FUNCTION_BLOCK Clock IMPLEMENTS Cyclic
VAR
	_Enable : BOOL;
	_Period : TIME;
	_Duty : LREAL := 0.5;
	switchTime : TIME;
	timer : TON;
	_Clock : BOOL;
END_VAR

METHOD PRIVATE CalcSwitchTime
switchTime := LREAL_TO_TIME(TIME_TO_LREAL(_Period) * _Duty);
END_METHOD

{attribute 'monitoring' := 'call'}
PROPERTY Clock : BOOL
GET
Clock := _Clock;
END_GET
END_PROPERTY

METHOD Cyclic
timer(IN := _Enable, PT := _Period);
IF (timer.Q) THEN
	timer(IN := FALSE);
	timer(IN := TRUE);
END_IF
_Clock := _Enable AND timer.ET >= switchTime;
END_METHOD

{attribute 'monitoring' := 'call'}
PROPERTY Duty : LREAL
GET
Duty := _Duty;
END_GET
SET
_Duty := Duty;
CalcSwitchTime();
END_SET
END_PROPERTY

{attribute 'monitoring' := 'call'}
PROPERTY Enable : BOOL
GET
Enable := _Enable;
END_GET
SET
_Enable := Enable;
END_SET
END_PROPERTY

{attribute 'monitoring' := 'call'}
PROPERTY Frequency : LREAL
GET
IF (_Period > T#0S) THEN
	Frequency := 1000/TIME_TO_LREAL(_Period);
ELSE
	Frequency := 0;
END_IF
END_GET
SET
IF (Frequency > 0) THEN
	_Period := LREAL_TO_TIME(1000/Frequency);
ELSE
	_Period := T#0S;
END_IF
CalcSwitchTime();
END_SET
END_PROPERTY

{attribute 'monitoring' := 'call'}
PROPERTY Period : TIME
GET
Period := _Period;
END_GET
SET
_Period := Period;
CalcSwitchTime();
END_SET
END_PROPERTY

END_FUNCTION_BLOCK

(* stored: Version 1.1.0.1
   POU Clock: Id {12e9d754-7a2e-04e4-151b-81bf53a123a4}, SpecialFunc None
   Method CalcSwitchTime: Id {eeb3fa65-90da-0834-10c0-64a9d6b20f5f}
   Property Clock: Id {94afcf8c-3fec-03bf-0ea5-551f99fbc25b}
   Get Get: Id {86ccfb57-1f88-0117-3a6c-95826046587c}
   Method Cyclic: Id {d126b246-8ccf-0404-1dbe-459eed47bff6}
   Property Duty: Id {62ad35f6-8917-03d8-1e82-2f52ccf6ca78}
   Get Get: Id {8de1ac67-05b7-0036-0652-56a889ec5cee}
   Set Set: Id {3b362bf6-5c6f-0809-0f27-e988aae87027}
   Property Enable: Id {6422a66f-fc11-03a1-3de3-f3d118b6b8d2}
   Get Get: Id {bbcdd0d0-b0bb-0fb1-3dd7-9ea84861c7f8}
   Set Set: Id {5d4d4c96-c66a-0ee5-2455-16a7b2586cfe}
   Property Frequency: Id {4bffecbf-5949-0b82-0871-84e2d868ed16}
   Get Get: Id {4748602e-ad65-03da-167f-a836679cba0a}
   Set Set: Id {22da3ccc-c4cc-06b8-171f-3c72e810f4b3}
   Property Period: Id {40003a89-ed2a-0499-316a-9142e6fbe1ba}
   Get Get: Id {1055d6d0-8094-0eb5-2db3-34798008d588}
   Set Set: Id {b3042076-8a6c-0519-1c2d-dd4b07d3ce04} *)
